FUNCTION_BLOCK Hutschienenmoped_6_DIA_DOUBLE_CLICK (* Service Interface Function Block Type *)
  (* Function: All Inputs *)
  (* Version 1.0, 2018-12-05, Jose Cabral *)
  (* Version 1.0_DOUBLE_CLICK, 2022-08-04, Franz Höpfinger, Unknown *)
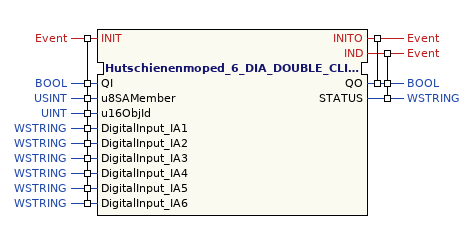
  EVENT_INPUT
    INIT WITH QI, u8SAMember, u16ObjId, DigitalInput_IA1, DigitalInput_IA2, DigitalInput_IA3, DigitalInput_IA4, DigitalInput_IA5, DigitalInput_IA6; (* Service Initialization *)
  END_EVENT
  EVENT_OUTPUT
    INITO WITH QO; (* Initialization Confirm *)
    IND WITH QO, STATUS; (* Indication from Resource *)
  END_EVENT
  VAR_INPUT
    QI : BOOL; (* Event Input Qualifier *)
    u8SAMember : USINT := 255; (* Dummy !, set to 255 if in doubt. 0 deactivates FB. *)
    u16ObjId : UINT := 65535; (* Dummy ! set to 65535 if in Doubt. 0 deactivates FB. *)
    DigitalInput_IA1 : WSTRING := "DigitalInput_IA1_DOUBLE_CLICK"; (* Identifier for Input 1 *)
    DigitalInput_IA2 : WSTRING := "DigitalInput_IA2_DOUBLE_CLICK"; (* Identifier for Input 2 *)
    DigitalInput_IA3 : WSTRING := "DigitalInput_IA3_DOUBLE_CLICK"; (* Identifier for Input 3 *)
    DigitalInput_IA4 : WSTRING := "DigitalInput_IA4_DOUBLE_CLICK"; (* Identifier for Input 4 *)
    DigitalInput_IA5 : WSTRING := "DigitalInput_IA5_DOUBLE_CLICK"; (* Identifier for Input 5 *)
    DigitalInput_IA6 : WSTRING := "DigitalInput_IA6_DOUBLE_CLICK"; (* Identifier for Input 6 *)
  END_VAR
  VAR_OUTPUT
    QO : BOOL; (* Event Output Qualifier *)
    STATUS : WSTRING; (* Service Status *)
  END_VAR
END_FUNCTION_BLOCK
